{attribute 'qualified_only'}
VAR_GLOBAL
	//Scanner to PLC
	//Load Tray Scanner
	In_Signal_Tray			: ST_BarcodeScanner;
	Out_Signal_Tray			: ST_BarcodeScanner;
	
	
	//Load Tray Scanner
	In_Signal_Conveyor		: ST_BarcodeScanner;
	Out_Signal_Conveyor		: ST_BarcodeScanner;

END_VAR

(* stored: Version 1.1.0.1, ProductVersion 3.1.4024.11
   GVL G_Scanner: Id {36bfca21-4f88-482f-a087-52dab6377d49} *)
